(********************************************************************************************)
(*							Beckhoff Automation Poland										*)
(*								FB_Blink_AS	 v1.1											*)
(*									9.11.2007												*)
(*						Blok funkcyjny zegara asynchronicznego								*)
(*__________________________________________________________________________________________*)

FUNCTION_BLOCK FB_Blink_AS
VAR_INPUT
	T1										:	TIME;				(*Czas, gdy wyjście przyjmuje wartość TRUE*)
	T0										:	TIME;				(*Czas, gdy wyjście przyjmuje wartość FALSE*)
END_VAR
VAR_OUTPUT
	Q										:	BOOL;				(*Wyjscie*)
END_VAR
VAR
	ton1									:	TON;
	ton2									:	TON;
END_VAR

ton1(IN:= NOT ton2.Q, PT:=T0);
Q:=ton1.Q;
ton2(IN:=ton1.Q , PT:=T1);

END_FUNCTION_BLOCK

(* stored: Version 1.1.0.1, ProductVersion 3.1.4026.13, FileIdentifier 354349ba032ae6df9cd99945d13dca08a722abd7, FileSignature 053efad7f5bf42ad4a11e027070c05b6bcacbf836d511d8688b2daaaba1a504ee7497ecb552ea98ec662a5776d5a3987d0e3addf2d3022be9912f6608970ccabfa3584ac49309613c387fa57dc0da4d32590807ec545c5192c5cc8904a14eb108ea7e6405f35b4d48a7f522a4214ce33b0dfa1538450ce88e57d4d4b81790c8f7fde1676c02b97b28918a4620f0529da7543ab5dd8fbe01ebcd267a23aa66df1ed0a9fb384ef1638582fe9cd2c5890794d3d432a42c27a9e70f0a97e51657e5772ea3786c7c20d824bd20d8908db5881c92bdbb4996e995682741036c217c6668ca877b7ded3dd545f36bcd2ac564812a073988c7705099a4ccf535f6df6f70f
   POU FB_Blink_AS: Id {308ba326-d075-48da-b682-df9e6ba1d528}, SpecialFunc None *)
